(* axis command structure *)
TYPE E_AxisCmd :
(
	Ax_Idle 		:= 0,// Axis command Referance 0 Axis Idle
	Ax_Init 		:= 1,// Axis command Referance 1 Initialize axis
	Ax_Enable 		:= 2,// Axis command Referance 2 Enable
	Ax_Disable 		:= 3,// Axis command Referance 3 Disable
	Ax_Reset 		:= 4,// Axis command Referance 4 Reset
	Ax_Hold 		:= 5,// Axis command Referance 5 Hold
	Ax_Home 		:= 6,// Axis command Referance 6 Home
	Ax_JogFwd 		:= 7,// Axis command Referance 7 Jog Forward
	Ax_JogRev 		:= 8,// Axis command Referance 8 Jog Reverse
	Ax_MoveRelative := 9,// Axis command Referance 9 Move axis relative
	Ax_MoveAbs 		:= 10,// Axis command Referance 11 Move absolute reverse
	Ax_MoveModulo 	:= 11,// Axis command Referance 11 Move Module
	Ax_MoveVeloFwd 	:= 12,// Axis command Referance 12 Move velocity forward
	Ax_MoveVeloRev 	:= 13,// Axis command Referance 13 Move velocity reverse
	Ax_HardStop 	:= 14,// Axis command Referance 14 hard stop or emergency stop
	Ax_SoftStop 	:= 15,// Axis command Referance 15 soft stop after motion command
	Ax_GearSlave 	:= 16,// Axis command Referance 16 gear axis as slave
	Ax_GearSlaveDyn	:= 17,// Axis command Referance 17 gear axis as slave dynamic
	Ax_GearOutSlave := 18,// Axis command Referance 18 gear out from Master axis 
	Ax_Maintenance	:= 50 // Axis Command referance 50 maintenance mode, axis enabled with no command active
);
END_TYPE

(* stored: Version 1.1.0.1, ProductVersion 3.1.4022.16
   EnumerationTextList E_AxisCmd: Id {8353c49c-d722-4c13-8e1d-2c20c8ac3f13} *)
